# B&R Automation Studio project CW2
Automation Studio 4.7.2.98

## Configuration CW2

CPU X20CP1382, AutomationRuntime C4.72, Build 4.1.2, Vc V4.72.0

### Task classes (Cpu.sw)
```
Cyclic#4:
  VVVFContro <- VVVFControl.prg
```

### Hardware
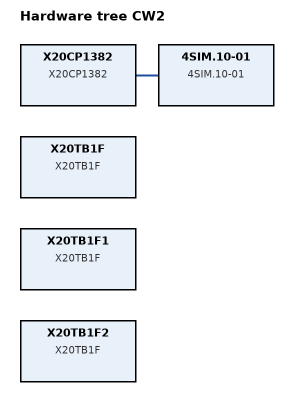
```
4SIM.10-01 : 4SIM.10-01 v1.3.0.0  [PLK1 -> X20CP1382.IF3 [Cable Type=PowerlinkCable, Length=10, Version=1.0.0.2]]
X20CP1382 : X20CP1382 v1.8.0.0  [X1 -> X1.SL; X2 -> X2.SL; X3 -> X3.SL]
  Module X1 (Type=X1, Virtual=true, Version=1.8.0.0)
    Connection (Connector=SS1, TargetModule=X20TB1F, TargetConnector=SS)
    Connection (Connector=SL, TargetModule=X20CP1382, TargetConnector=X1)
  Module X2 (Type=X2, Virtual=true, Version=1.8.0.0)
    Connection (Connector=SS1, TargetModule=X20TB1F1, TargetConnector=SS)
    Connection (Connector=SL, TargetModule=X20CP1382, TargetConnector=X2)
  Module X3 (Type=X3, Virtual=true, Version=1.8.0.0)
    Connection (Connector=SS1, TargetModule=X20TB1F2, TargetConnector=SS)
    Connection (Connector=SL, TargetModule=X20CP1382, TargetConnector=X3)
  Connector IF2:
    ActivateDevice = 1
  ConfigurationID = CW2_CW2
  Simulation = 1
X20TB1F : X20TB1F v1.0.0.0
X20TB1F1 : X20TB1F v1.0.0.0
X20TB1F2 : X20TB1F v1.0.0.0
```

### IoMap.iom - X20CP1382/IoMap.iom
```iecst
VAR_CONFIG
	::VVVFContro:SB2 AT %IX."4SIM.10-01".DigitalInput01;
	::VVVFContro:SF AT %IX."4SIM.10-01".DigitalInput02;
	::VVVFContro:SB3 AT %IX."4SIM.10-01".DigitalInput03;
	::VVVFContro:SB4 AT %IX."4SIM.10-01".DigitalInput04;
	::VVVFContro:SB5 AT %IX."4SIM.10-01".DigitalInput05;
	::VVVFContro:HL1 AT %QX."4SIM.10-01".DigitalOutput01;
	::VVVFContro:HL2 AT %QX."4SIM.10-01".DigitalOutput05;
	::VVVFContro:HL3 AT %QX."4SIM.10-01".DigitalOutput03;
END_VAR
```

## Logical view

### Program Logical/VVVFControl (IEC)

#### Cyclic.ld - Cyclic code
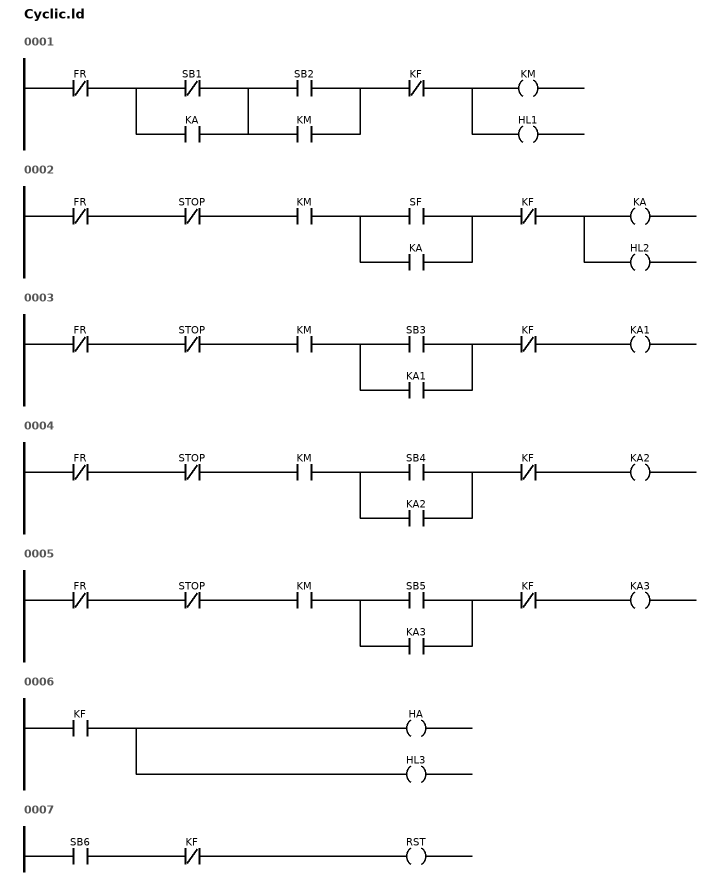
Ladder, written as Structured Text:
```iecst
PROGRAM _CYCLIC
VAR
    _p1 : BOOL;
    _p2 : BOOL;
END_VAR
(* Network 1 *)
_p1 := NOT FR AND (NOT SB1 OR KA) AND (SB2 OR KM) AND NOT KF;
KM := _p1;
HL1 := _p1;

(* Network 2 *)
_p2 := NOT FR AND NOT STOP AND KM AND (SF OR KA) AND NOT KF;
KA := _p2;
HL2 := _p2;

(* Network 3 *)
KA1 := NOT FR AND NOT STOP AND KM AND (SB3 OR KA1) AND NOT KF;

(* Network 4 *)
KA2 := NOT FR AND NOT STOP AND KM AND (SB4 OR KA2) AND NOT KF;

(* Network 5 *)
KA3 := NOT FR AND NOT STOP AND KM AND (SB5 OR KA3) AND NOT KF;

(* Network 6 *)
HA := KF;
HL3 := KF;

(* Network 7 *)
RST := SB6 AND NOT KF;
END_PROGRAM
```

#### Variables.var - Local variables
```iecst
VAR
	SB1 : BOOL; (*power off buttom*)
	SB2 : BOOL; (*power on buttom*)
	FR : BOOL; (*overload relay*)
	KF : BOOL; (*fault flag*)
	KM : BOOL; (*power on contactor*)
	HL1 : BOOL; (*power on indicator*)
	KA : BOOL; (*control relay for start*)
	STOP : BOOL; (*motor stop*)
	SF : BOOL; (*motor start buttom*)
	HL2 : BOOL; (*motor moving indicator*)
	SB3 : BOOL; (*speed 1 push buttom*)
	KA1 : BOOL; (*speed 1*)
	SB4 : BOOL; (*speed 2 push buttom*)
	KA2 : BOOL; (*speed 2*)
	KA3 : BOOL; (*speed 3*)
	SB5 : BOOL; (*speed 3 push buttom*)
	HA : BOOL; (*fault alarm*)
	HL3 : BOOL; (*fault indicator light*)
	SB6 : BOOL; (*reset switch*)
	RST : BOOL; (*reset flag*)
END_VAR
```

Listed in the project but not available here: Logical/Global.typ, Logical/Global.var, Logical/Libraries, Logical/VVVFControl/Init.ld, Logical/VVVFControl/Exit.ld, Logical/VVVFControl/Types.typ
